// Mitsubishi GX Works2 project: exam08_modbus_master   PLC: FX1N/FX1NC

PROGRAM MAIN
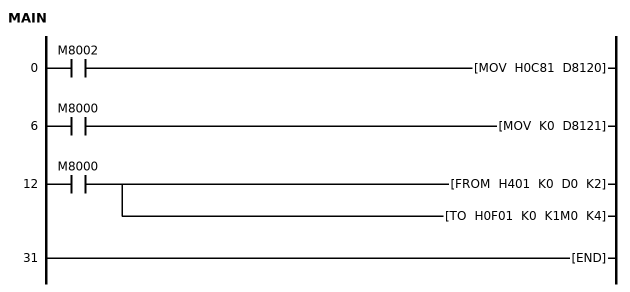
0     LD      M8002
      MOV     H0C81 D8120
6     LD      M8000
      MOV     K0 D8121
12    LD      M8000
      FROM    H401 K0 D0 K2
      TO      H0F01 K0 K1M0 K4
31    END
END_PROGRAM
